{attribute 'qualified_only'}
{attribute 'strict'}
TYPE State_Dispenser :
(
	Off,
	Reset, 
	Reset_done,
	Power, 
	Ready, 
	Dispensing,
	Done,
	Wait
);
END_TYPE

(* stored: Version 1.1.0.1, ProductVersion 3.1.4024.12
   DUT State_Dispenser: Id {2e85bf90-75b0-49bf-acdd-cd88a9e3c418} *)
